{attribute addProperty BoxType "EL1258-0010-0017"}
{attribute addProperty Id "MTI_Inputs_1x_ChannelAT %I*ARRAY[0..21] OF MTI_Inputs_1x_Channel_43566A27768960MTI_Outputs_ChannelAT %Q*ARRAY[0..7] OF MTI_Outputs_Channel_0FF822EF256320WcStateAT %I*WcState_98A4DF7520.250InfoDataAT %I*InfoData_0BDED7BF144180"}
{attribute addProperty CRC "8436216"}
{attribute addProperty SizeInBites "1170"}
{attribute addProperty SizeInBytes "146.25"}
TYPE EL1258_62C936BD :
STRUCT
	{attribute addProperty Name "MTI_Inputs_1x_Channel"}
	MTI_Inputs_1x_Channel : ARRAY[0..21] OF MTI_Inputs_1x_Channel_43566A27;
	{attribute addProperty Name "MTI_Outputs_Channel"}
	MTI_Outputs_Channel : ARRAY[0..7] OF MTI_Outputs_Channel_0FF822EF;
	{attribute addProperty Name "WcState"}
	WcState : WcState_98A4DF75;
	{attribute addProperty Name "InfoData"}
	InfoData : InfoData_0BDED7BF;
END_STRUCT
END_TYPE

(* stored: Version 1.2.0.0, ProductVersion 3.1.4024.9
   DUT EL1258_62C936BD: Id {c97d2a52-8149-477f-ace7-23d4ff5d1773} *)
